{attribute 'qualified_only'}
{attribute 'strict'}
{attribute 'to_string'}
TYPE
ST105_Pnp_e :
(
    RESET := 0, // Reset

    INIT := 100, // Initialisieren 
    Init_HomeVertical,
    Init_VerticalDown,
    Init_RobotRaiseStartFlag,
    Init_RobotFallStartFlag,
    Init_check_if_pces_handled,

    READY := 999,  // READY to Start, Init Done 
    START := 1000, // Start Zyklisch
    MOVER_FREE_OP, // Ab here, operation without mover can be done

    wait_on_feeder, // wait on feeder to be ready
    push_up_casing, // push up the casing (gehäuse)
    Robot_Pick,     // send pick signal to the robot
    Robot_wait_picked_falling,
    pusher_down,

    waitOnMover,     // wait until the mover is there
    MOVER_NEEDED_OP, // Since here, a mover in position is needed to perform the action

    Robot_place, // send place signal to the robot
    Robot_wait_placed_falling,

    SYNC_MOVER_LEAVE, // MoverMan need to take the mover
    DONE := 8000,     // Ablauf beendet 
    ERROR := 9000,    // Fehler 
    _max
);
END_TYPE

(* stored: Version 1.1.0.1, ProductVersion 3.1.4024.6
   EnumerationTextList ST105_Pnp_e: Id {3b670f93-e452-4645-96c8-fd6060492713} *)
